TYPE ST_COMMAND :
STRUCT
	command:INT;
	distance:LREAL;
	direction:INT;
	acc:LREAL;
	jerk:LREAL;
	spd:LREAL;
END_STRUCT
END_TYPE

(* stored: Version 1.1.0.1, ProductVersion 3.1.4024.12
   DUT ST_COMMAND: Id {16b13aeb-8fe5-4128-82f5-02317289abe7} *)
